FUNCTION Vector_Magnitude : BOOL
VAR_INPUT
	IN : REFERENCE TO Matrix;
END_VAR
VAR_OUTPUT
	Res : LREAL;
END_VAR
VAR
	Sum : LREAL;
	I : UINT;
END_VAR

IF NOT(IN.IsVector) OR IN.IsEmpty THEN
	Res := 0;
	Vector_Magnitude := FALSE;
	RETURN;
END_IF

Vector_Magnitude := TRUE;
Sum := 0;

FOR I := 0 TO IN.Length-1 DO
	Sum := Sum + IN.GetI(I) * IN.GetI(I);
END_FOR

Res := SQRT(Sum);

END_FUNCTION

(* stored: Version 1.1.0.1, ProductVersion 3.1.4024.9
   POU Vector_Magnitude: Id {196a9e75-9374-02ba-0429-dfa5e7be03f4}, SpecialFunc None *)
